PROGRAM Circuito_L8
VAR_INPUT
	Modo_Calibrar_L8: BOOL;
END_VAR
VAR
		fbBomba_L8 :Equipo_Motor_ATV320;
		ControlValv_ioLink_V1:ControlValv_ioLink;
		ControlValv_ioLink_V2: ControlValv_ioLink;
		ControlValv_ioLink_V3: ControlValv_ioLink;
		ControlValv_ioLink_V4: ControlValv_ioLink;
		Falla_L8_V1:BOOL;
		Falla_L8_V2:BOOL;
		Falla_L8_V3:BOOL;
		Falla_L8_V4:BOOL;
	Balanza_PU2_WT8: Balanza;
		dHS:DINT;
		TOF_calibradoIBC: TOF;
		PID_L8_SP:REAL;
		PID_L8_auto:BOOL;
		PID_L8_reset:BOOL;
		PID_L8_manual:REAL;
		PID_L8_bMuerta:REAL := 5;
		PID_L8_Kp:REAL := 0.1;
		PID_L8_Ti:REAL := 100;
		PID_L8_PV:REAL;
		Dosis_L8	:REAL;
		TiempoInyeccion_L8	:DINT;
		Peso	:REAL;
		Offset_L8:REAL;
		Inyeccion_L8:BOOL;
		Volumen_L8:REAL;
		Calculo_caudal_L8: Calculo_caudal;
		CorrecionCaudalxOffset_L8: CorrecionCaudalxOffset;
		tInyeccion: TON;
		Total :REAL;
		Totalant	:REAL;
		auxIniCal:BOOL;
		AuxVol:REAL;
		CA2_L8_V1_CmdA_Man :BOOL;
		CA2_L8_V4_CmdA_Man :BOOL;
		TDemoraInyectar: TON;
		SetDemoraInyeccion: REAL;
		Tiempo_seg_to_TIME_DemoraInyec: Tiempo_seg_to_TIME;
		AuxTDemoraInyec: TIME;
		PID_L8: FB_PID;		
		Tiempo_TIME_to_seg_InyCal: Tiempo_TIME_to_seg;
		AuxInyCal:TIME;	
		IniTotalFT2:REAL;
		Auxconsumo:REAL;
	ProductoAsociado: STRING;
	Lavagem_Circuito08: Lavagem;
	BasicPID_L8: FB_BasicPID;
	Teste: BOOL;
	Filtro:Filtro2;
	TON_StartBomba: TON;
END_VAR

VAR PERSISTENT
	UltimaCalibracao	:UDINT;	//Data e hora da ultima calibração
END_VAR
VAR // added by the converter: edge detectors and wires of the graphical bodies
    _w1, _w2, _w3, _w4, _w5, _w6, _w7, _w8, _w9, _w10, _w11, _w12, _w13 : BOOL;
    _ft1 : F_TRIG;
    _rt1, _rt2, _rt3 : R_TRIG;
END_VAR

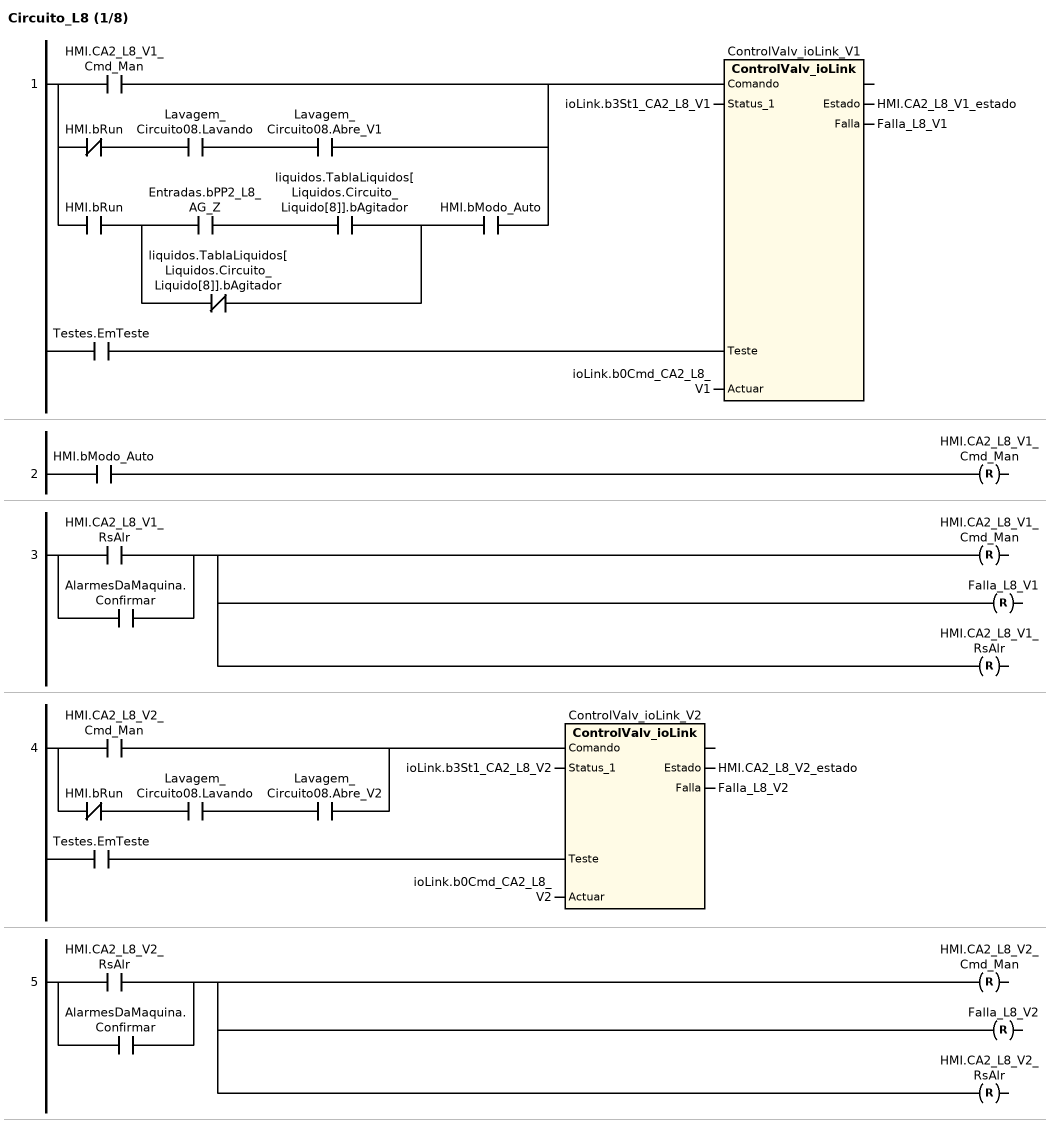
// NETWORK 1
ControlValv_ioLink_V1(
    Comando := HMI.CA2_L8_V1_Cmd_Man OR NOT HMI.bRun AND Lavagem_Circuito08.Lavando AND Lavagem_Circuito08.Abre_V1 OR HMI.bRun AND (Entradas.bPP2_L8_AG_Z AND (liquidos.TablaLiquidos[Liquidos.Circuito_Liquido[8]].bAgitador) OR NOT (liquidos.TablaLiquidos[Liquidos.Circuito_Liquido[8]].bAgitador)) AND HMI.bModo_Auto,
    Status_1 := ioLink.b3St1_CA2_L8_V1,
    Teste := Testes.EmTeste,
    Actuar := ioLink.b0Cmd_CA2_L8_V1,
    Estado => HMI.CA2_L8_V1_estado,
    Falla => Falla_L8_V1); // ControlValv_ioLink

// NETWORK 2
HMI.CA2_L8_V1_Cmd_Man R= HMI.bModo_Auto;

// NETWORK 3
_w1 := HMI.CA2_L8_V1_RsAlr OR AlarmesDaMaquina.Confirmar;
HMI.CA2_L8_V1_Cmd_Man R= _w1;
Falla_L8_V1 R= _w1;
HMI.CA2_L8_V1_RsAlr R= _w1;

// NETWORK 4
ControlValv_ioLink_V2(
    Comando := HMI.CA2_L8_V2_Cmd_Man OR NOT HMI.bRun AND Lavagem_Circuito08.Lavando AND Lavagem_Circuito08.Abre_V2,
    Status_1 := ioLink.b3St1_CA2_L8_V2,
    Teste := Testes.EmTeste,
    Actuar := ioLink.b0Cmd_CA2_L8_V2,
    Estado => HMI.CA2_L8_V2_estado,
    Falla => Falla_L8_V2); // ControlValv_ioLink

// NETWORK 5
_w2 := HMI.CA2_L8_V2_RsAlr OR AlarmesDaMaquina.Confirmar;
HMI.CA2_L8_V2_Cmd_Man R= _w2;
Falla_L8_V2 R= _w2;
HMI.CA2_L8_V2_RsAlr R= _w2;

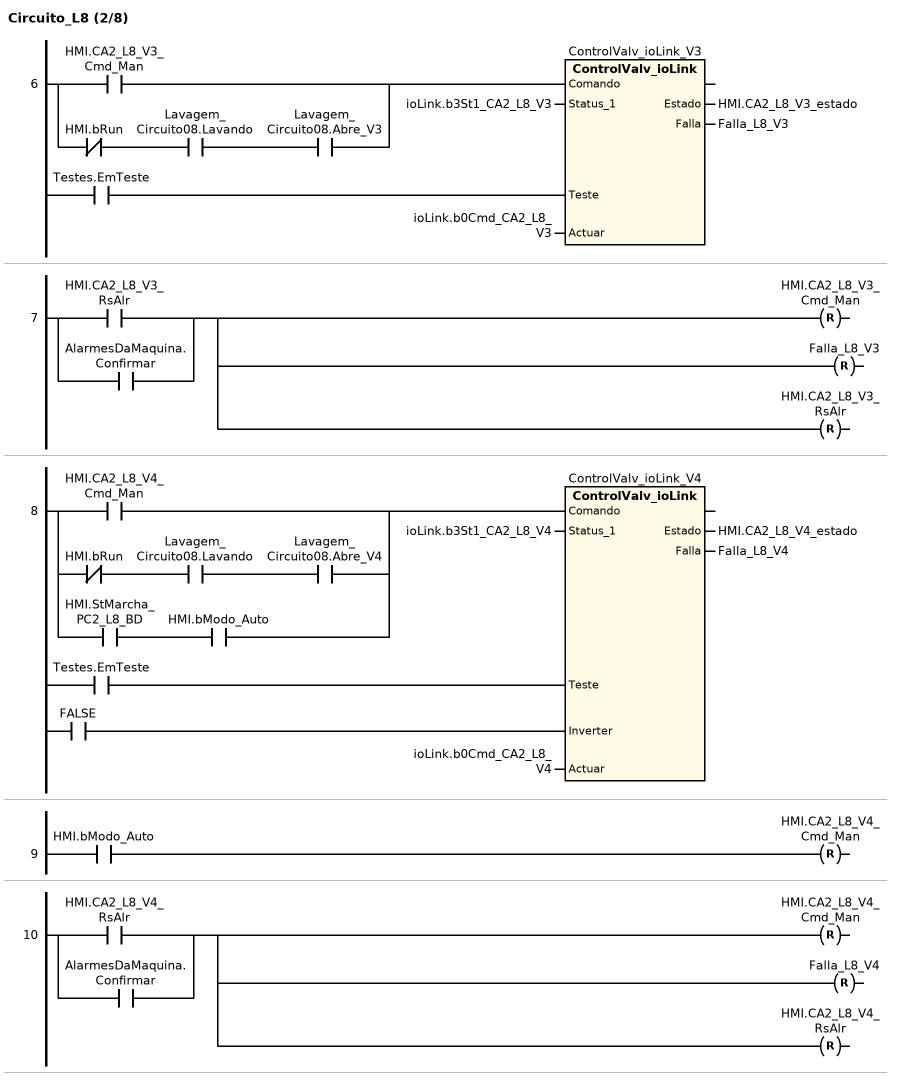
// NETWORK 6
ControlValv_ioLink_V3(
    Comando := HMI.CA2_L8_V3_Cmd_Man OR NOT HMI.bRun AND Lavagem_Circuito08.Lavando AND Lavagem_Circuito08.Abre_V3,
    Status_1 := ioLink.b3St1_CA2_L8_V3,
    Teste := Testes.EmTeste,
    Actuar := ioLink.b0Cmd_CA2_L8_V3,
    Estado => HMI.CA2_L8_V3_estado,
    Falla => Falla_L8_V3); // ControlValv_ioLink

// NETWORK 7
_w3 := HMI.CA2_L8_V3_RsAlr OR AlarmesDaMaquina.Confirmar;
HMI.CA2_L8_V3_Cmd_Man R= _w3;
Falla_L8_V3 R= _w3;
HMI.CA2_L8_V3_RsAlr R= _w3;

// NETWORK 8
ControlValv_ioLink_V4(
    Comando := HMI.CA2_L8_V4_Cmd_Man OR NOT HMI.bRun AND Lavagem_Circuito08.Lavando AND Lavagem_Circuito08.Abre_V4 OR HMI.StMarcha_PC2_L8_BD AND HMI.bModo_Auto,
    Status_1 := ioLink.b3St1_CA2_L8_V4,
    Teste := Testes.EmTeste,
    Inverter := FALSE,
    Actuar := ioLink.b0Cmd_CA2_L8_V4,
    Estado => HMI.CA2_L8_V4_estado,
    Falla => Falla_L8_V4); // ControlValv_ioLink

// NETWORK 9
HMI.CA2_L8_V4_Cmd_Man R= HMI.bModo_Auto;

// NETWORK 10
_w4 := HMI.CA2_L8_V4_RsAlr OR AlarmesDaMaquina.Confirmar;
HMI.CA2_L8_V4_Cmd_Man R= _w4;
Falla_L8_V4 R= _w4;
HMI.CA2_L8_V4_RsAlr R= _w4;

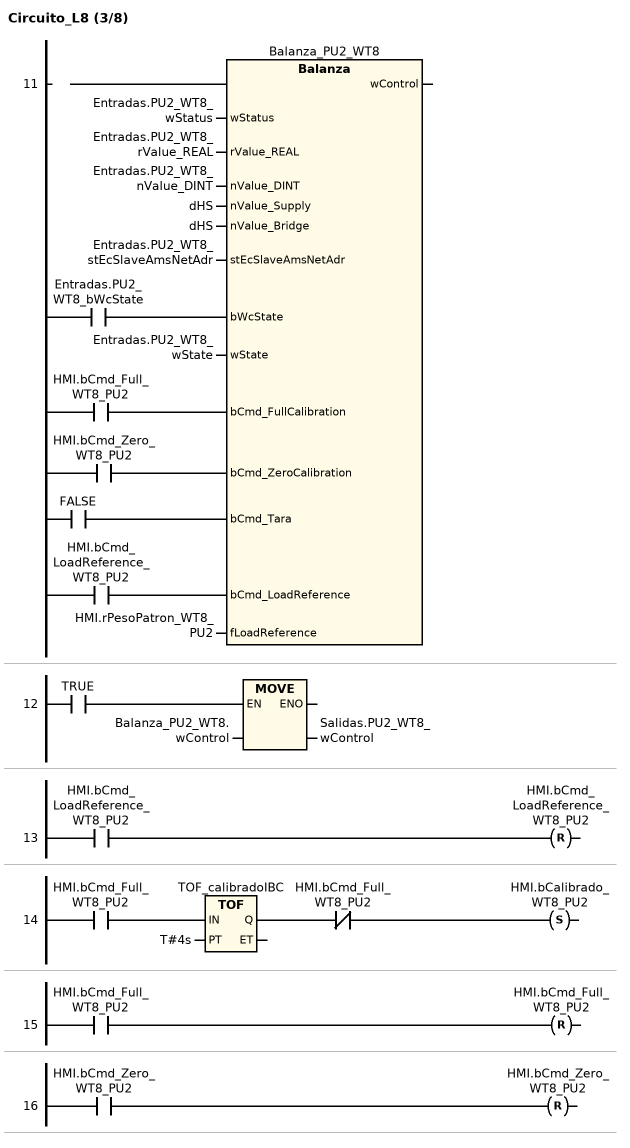
// NETWORK 11
Balanza_PU2_WT8(
    wStatus := Entradas.PU2_WT8_wStatus,
    rValue_REAL := Entradas.PU2_WT8_rValue_REAL,
    nValue_DINT := Entradas.PU2_WT8_nValue_DINT,
    nValue_Supply := dHS,
    nValue_Bridge := dHS,
    stEcSlaveAmsNetAdr := Entradas.PU2_WT8_stEcSlaveAmsNetAdr,
    bWcState := Entradas.PU2_WT8_bWcState,
    wState := Entradas.PU2_WT8_wState,
    bCmd_FullCalibration := HMI.bCmd_Full_WT8_PU2,
    bCmd_ZeroCalibration := HMI.bCmd_Zero_WT8_PU2,
    bCmd_Tara := FALSE,
    bCmd_LoadReference := HMI.bCmd_LoadReference_WT8_PU2,
    fLoadReference := HMI.rPesoPatron_WT8_PU2); // Balanza

// NETWORK 12
Salidas.PU2_WT8_wControl := Balanza_PU2_WT8.wControl;

// NETWORK 13
HMI.bCmd_LoadReference_WT8_PU2 R= HMI.bCmd_LoadReference_WT8_PU2;

// NETWORK 14
TOF_calibradoIBC(IN := HMI.bCmd_Full_WT8_PU2, PT := T#4s); // TOF
HMI.bCalibrado_WT8_PU2 S= TOF_calibradoIBC.Q AND NOT HMI.bCmd_Full_WT8_PU2;

// NETWORK 15
HMI.bCmd_Full_WT8_PU2 R= HMI.bCmd_Full_WT8_PU2;

// NETWORK 16
HMI.bCmd_Zero_WT8_PU2 R= HMI.bCmd_Zero_WT8_PU2;

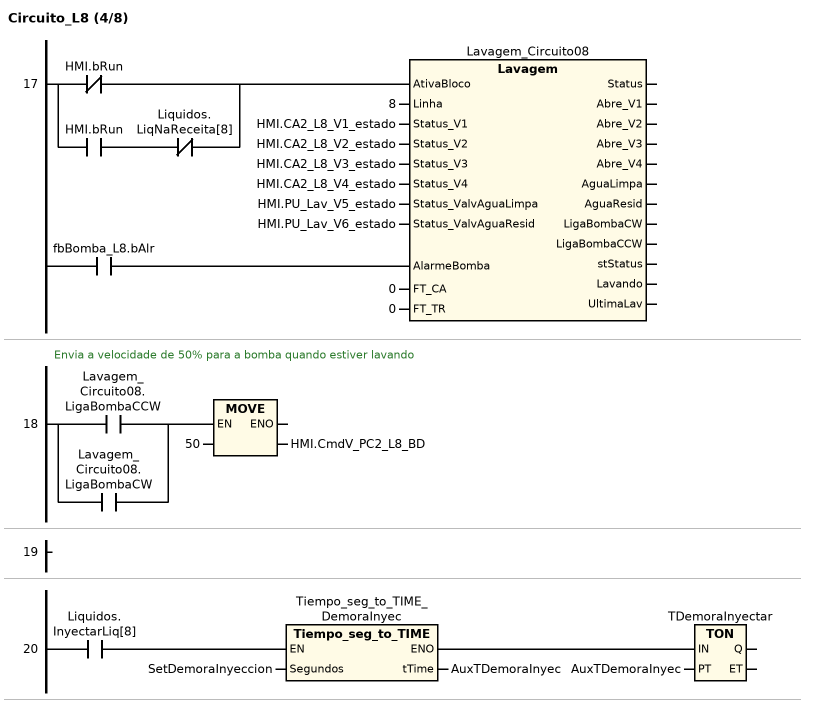
// NETWORK 17
Lavagem_Circuito08(
    AtivaBloco := NOT HMI.bRun OR HMI.bRun AND NOT Liquidos.LiqNaReceita[8],
    Linha := 8,
    Status_V1 := HMI.CA2_L8_V1_estado,
    Status_V2 := HMI.CA2_L8_V2_estado,
    Status_V3 := HMI.CA2_L8_V3_estado,
    Status_V4 := HMI.CA2_L8_V4_estado,
    Status_ValvAguaLimpa := HMI.PU_Lav_V5_estado,
    Status_ValvAguaResid := HMI.PU_Lav_V6_estado,
    AlarmeBomba := fbBomba_L8.bAlr,
    FT_CA := 0,
    FT_TR := 0); // Lavagem

// NETWORK 18
// Envia a velocidade de 50% para a bomba quando estiver lavando
IF Lavagem_Circuito08.LigaBombaCCW OR Lavagem_Circuito08.LigaBombaCW THEN HMI.CmdV_PC2_L8_BD := 50; END_IF

// NETWORK 19

// NETWORK 20
_w5 := Liquidos.InyectarLiq[8];
IF _w5 THEN
    Tiempo_seg_to_TIME_DemoraInyec(Segundos := SetDemoraInyeccion, tTime => AuxTDemoraInyec); // Tiempo_seg_to_TIME
END_IF
TDemoraInyectar(IN := _w5, PT := AuxTDemoraInyec); // TON

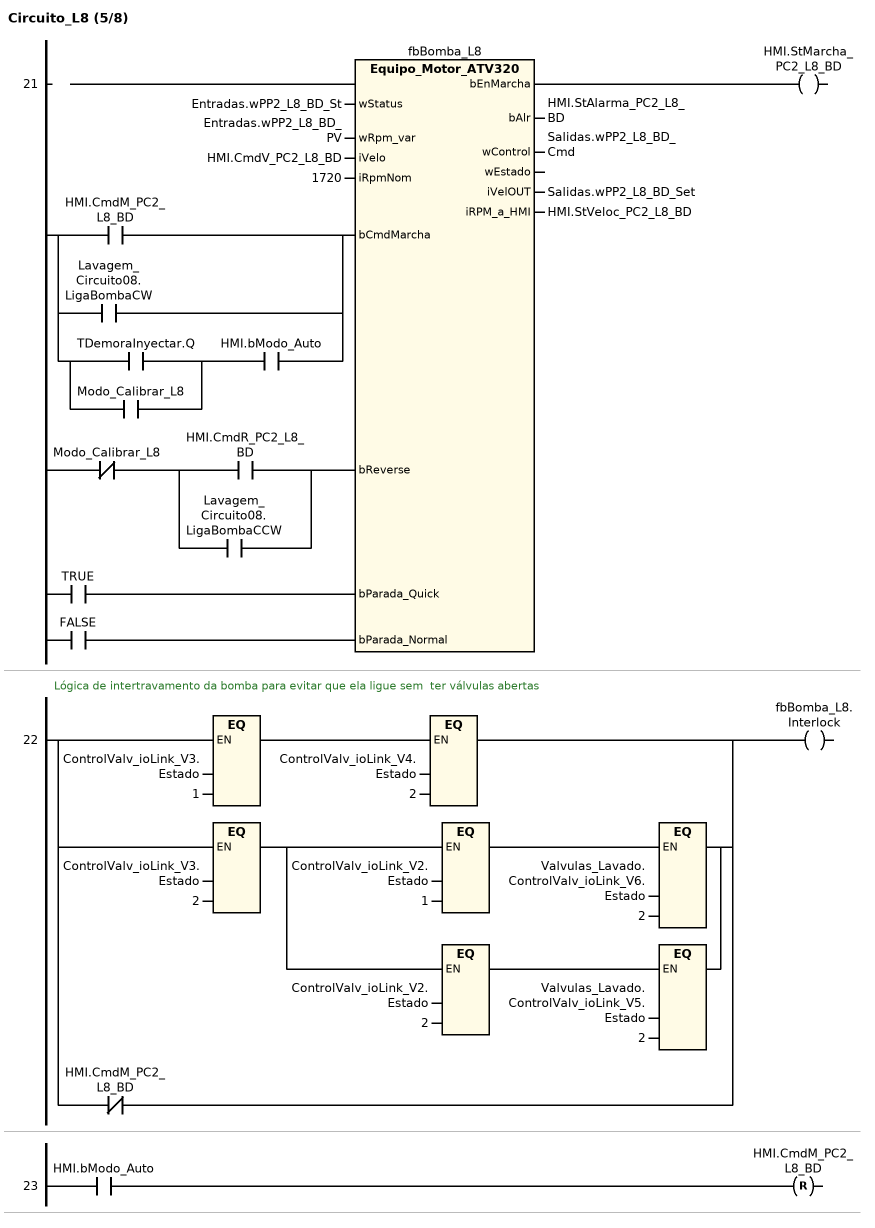
// NETWORK 21
fbBomba_L8(
    wStatus := Entradas.wPP2_L8_BD_St,
    wRpm_var := Entradas.wPP2_L8_BD_PV,
    iVelo := HMI.CmdV_PC2_L8_BD,
    iRpmNom := 1720,
    bCmdMarcha := HMI.CmdM_PC2_L8_BD OR Lavagem_Circuito08.LigaBombaCW OR (TDemoraInyectar.Q OR Modo_Calibrar_L8) AND HMI.bModo_Auto,
    bReverse := NOT Modo_Calibrar_L8 AND (HMI.CmdR_PC2_L8_BD OR Lavagem_Circuito08.LigaBombaCCW),
    bParada_Quick := TRUE,
    bParada_Normal := FALSE,
    bAlr => HMI.StAlarma_PC2_L8_BD,
    wControl => Salidas.wPP2_L8_BD_Cmd,
    iVelOUT => Salidas.wPP2_L8_BD_Set,
    iRPM_a_HMI => HMI.StVeloc_PC2_L8_BD); // Equipo_Motor_ATV320
HMI.StMarcha_PC2_L8_BD := fbBomba_L8.bEnMarcha;

// NETWORK 22
// Lógica de intertravamento da bomba para evitar que ela ligue sem  ter válvulas abertas
_w6 := NOT HMI.CmdM_PC2_L8_BD;
IF NOT _w6 THEN
    _w7 := ControlValv_ioLink_V3.Estado = 2;
    _w6 := ControlValv_ioLink_V3.Estado = 1 AND ControlValv_ioLink_V4.Estado = 2 OR (_w7 AND ControlValv_ioLink_V2.Estado = 1 AND Valvulas_Lavado.ControlValv_ioLink_V6.Estado = 2 OR _w7 AND ControlValv_ioLink_V2.Estado = 2 AND Valvulas_Lavado.ControlValv_ioLink_V5.Estado = 2);
END_IF
fbBomba_L8.Interlock := _w6;

// NETWORK 23
HMI.CmdM_PC2_L8_BD R= HMI.bModo_Auto;

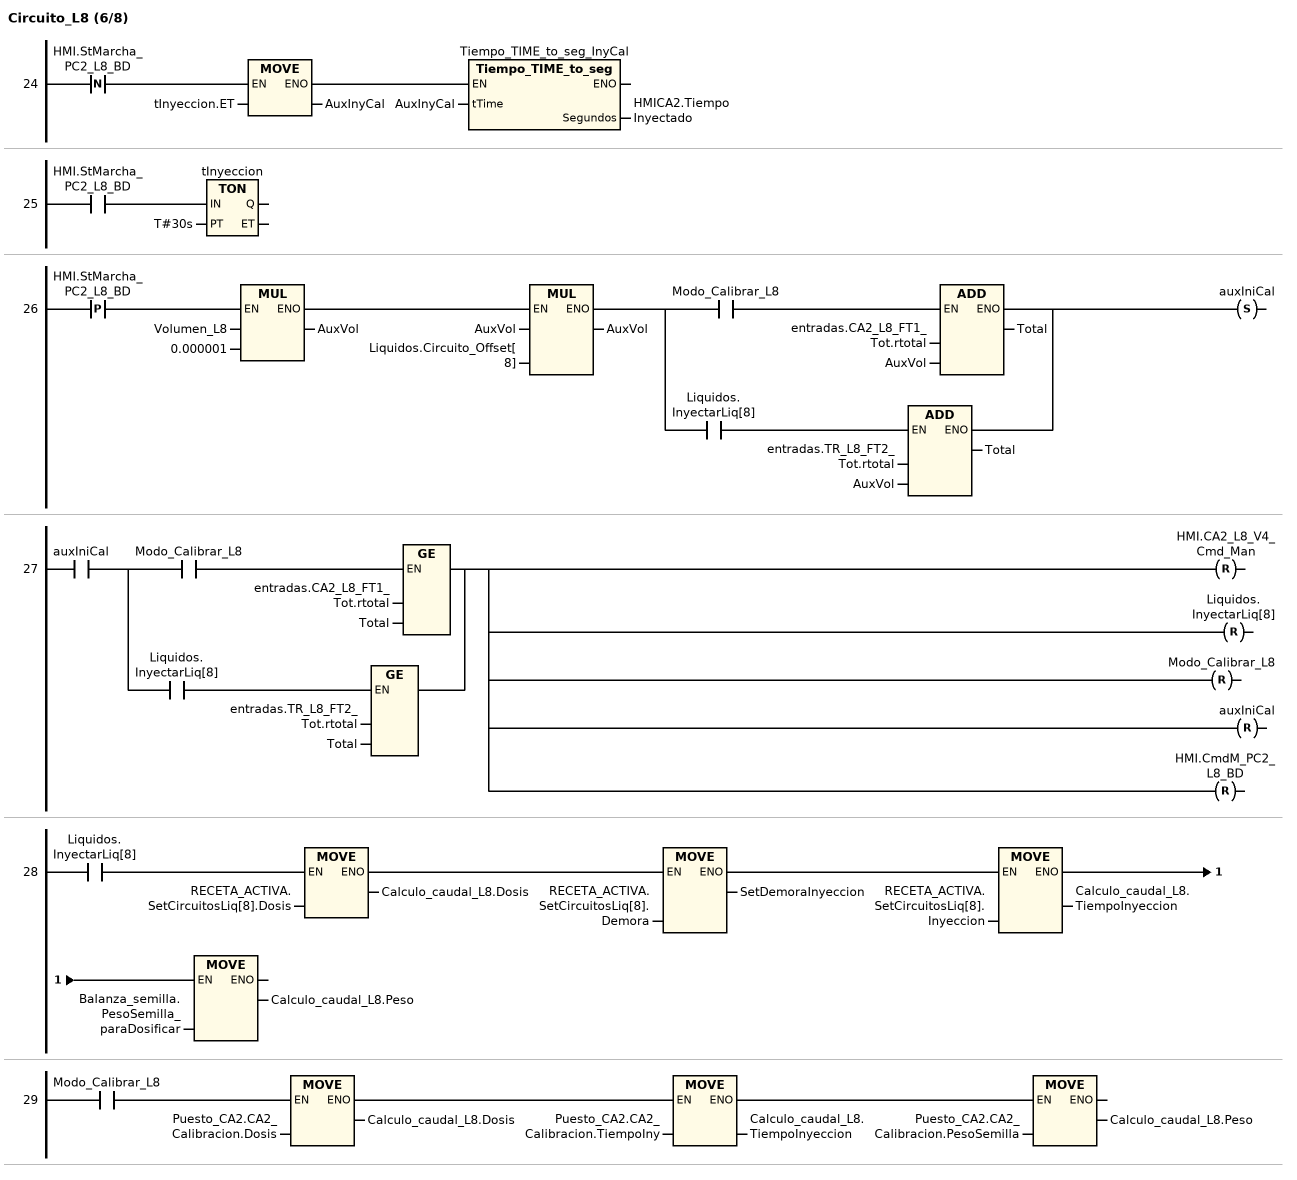
// NETWORK 24
_ft1(CLK := HMI.StMarcha_PC2_L8_BD);
_w8 := _ft1.Q;
IF _w8 THEN AuxInyCal := tInyeccion.ET; END_IF
IF _w8 THEN
    Tiempo_TIME_to_seg_InyCal(tTime := AuxInyCal, Segundos => HMICA2.TiempoInyectado); // Tiempo_TIME_to_seg
END_IF

// NETWORK 25
tInyeccion(IN := HMI.StMarcha_PC2_L8_BD, PT := T#30s); // TON

// NETWORK 26
_rt1(CLK := HMI.StMarcha_PC2_L8_BD);
_w9 := _rt1.Q;
IF _w9 THEN AuxVol := Volumen_L8 * 0.000001; END_IF
IF _w9 THEN AuxVol := AuxVol * Liquidos.Circuito_Offset[8]; END_IF
IF _w9 AND Modo_Calibrar_L8 THEN Total := entradas.CA2_L8_FT1_Tot.rtotal + AuxVol; END_IF
IF _w9 AND Liquidos.InyectarLiq[8] THEN Total := entradas.TR_L8_FT2_Tot.rtotal + AuxVol; END_IF
auxIniCal S= _w9 AND Modo_Calibrar_L8 OR _w9 AND Liquidos.InyectarLiq[8];

// NETWORK 27
_w10 := auxIniCal AND Modo_Calibrar_L8 AND entradas.CA2_L8_FT1_Tot.rtotal >= Total OR auxIniCal AND Liquidos.InyectarLiq[8] AND entradas.TR_L8_FT2_Tot.rtotal >= Total;
HMI.CA2_L8_V4_Cmd_Man R= _w10;
Liquidos.InyectarLiq[8] R= _w10;
Modo_Calibrar_L8 R= _w10;
auxIniCal R= _w10;
HMI.CmdM_PC2_L8_BD R= _w10;

// NETWORK 28
_w11 := Liquidos.InyectarLiq[8];
IF _w11 THEN Calculo_caudal_L8.Dosis := RECETA_ACTIVA.SetCircuitosLiq[8].Dosis; END_IF
IF _w11 THEN SetDemoraInyeccion := RECETA_ACTIVA.SetCircuitosLiq[8].Demora; END_IF
IF _w11 THEN Calculo_caudal_L8.TiempoInyeccion := RECETA_ACTIVA.SetCircuitosLiq[8].Inyeccion; END_IF
IF _w11 THEN Calculo_caudal_L8.Peso := Balanza_semilla.PesoSemilla_paraDosificar; END_IF

// NETWORK 29
_w12 := Modo_Calibrar_L8;
IF _w12 THEN Calculo_caudal_L8.Dosis := Puesto_CA2.CA2_Calibracion.Dosis; END_IF
IF _w12 THEN Calculo_caudal_L8.TiempoInyeccion := Puesto_CA2.CA2_Calibracion.TiempoIny; END_IF
IF _w12 THEN Calculo_caudal_L8.Peso := Puesto_CA2.CA2_Calibracion.PesoSemilla; END_IF

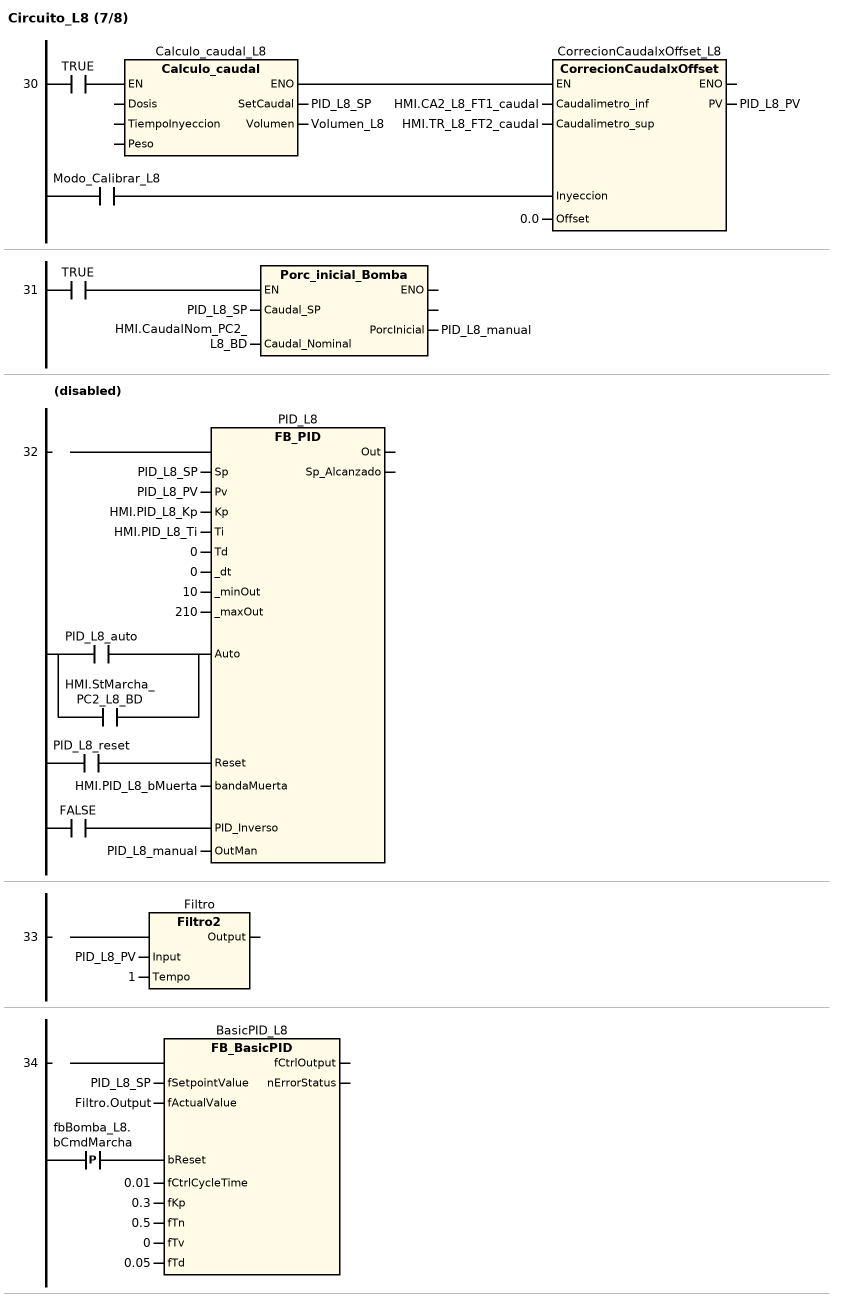
// NETWORK 30
Calculo_caudal_L8(SetCaudal => PID_L8_SP, Volumen => Volumen_L8); // Calculo_caudal
CorrecionCaudalxOffset_L8(
    Caudalimetro_inf := HMI.CA2_L8_FT1_caudal,
    Caudalimetro_sup := HMI.TR_L8_FT2_caudal,
    Inyeccion := Modo_Calibrar_L8,
    Offset := 0.0,
    PV => PID_L8_PV); // CorrecionCaudalxOffset

// NETWORK 31
Porc_inicial_Bomba(Caudal_SP := PID_L8_SP, Caudal_Nominal := HMI.CaudalNom_PC2_L8_BD, PorcInicial => PID_L8_manual);

// NETWORK 32 (disabled)
// PID_L8(
//     Sp := PID_L8_SP,
//     Pv := PID_L8_PV,
//     Kp := HMI.PID_L8_Kp,
//     Ti := HMI.PID_L8_Ti,
//     Td := 0,
//     _dt := 0,
//     _minOut := 10,
//     _maxOut := 210,
//     Auto := PID_L8_auto OR HMI.StMarcha_PC2_L8_BD,
//     Reset := PID_L8_reset,
//     bandaMuerta := HMI.PID_L8_bMuerta,
//     PID_Inverso := FALSE,
//     OutMan := PID_L8_manual); // FB_PID

// NETWORK 33
Filtro(Input := PID_L8_PV, Tempo := 1); // Filtro2

// NETWORK 34
_rt2(CLK := fbBomba_L8.bCmdMarcha);
BasicPID_L8(
    fSetpointValue := PID_L8_SP,
    fActualValue := Filtro.Output,
    bReset := _rt2.Q,
    fCtrlCycleTime := 0.01,
    fKp := 0.3,
    fTn := 0.5,
    fTv := 0,
    fTd := 0.05); // FB_BasicPID

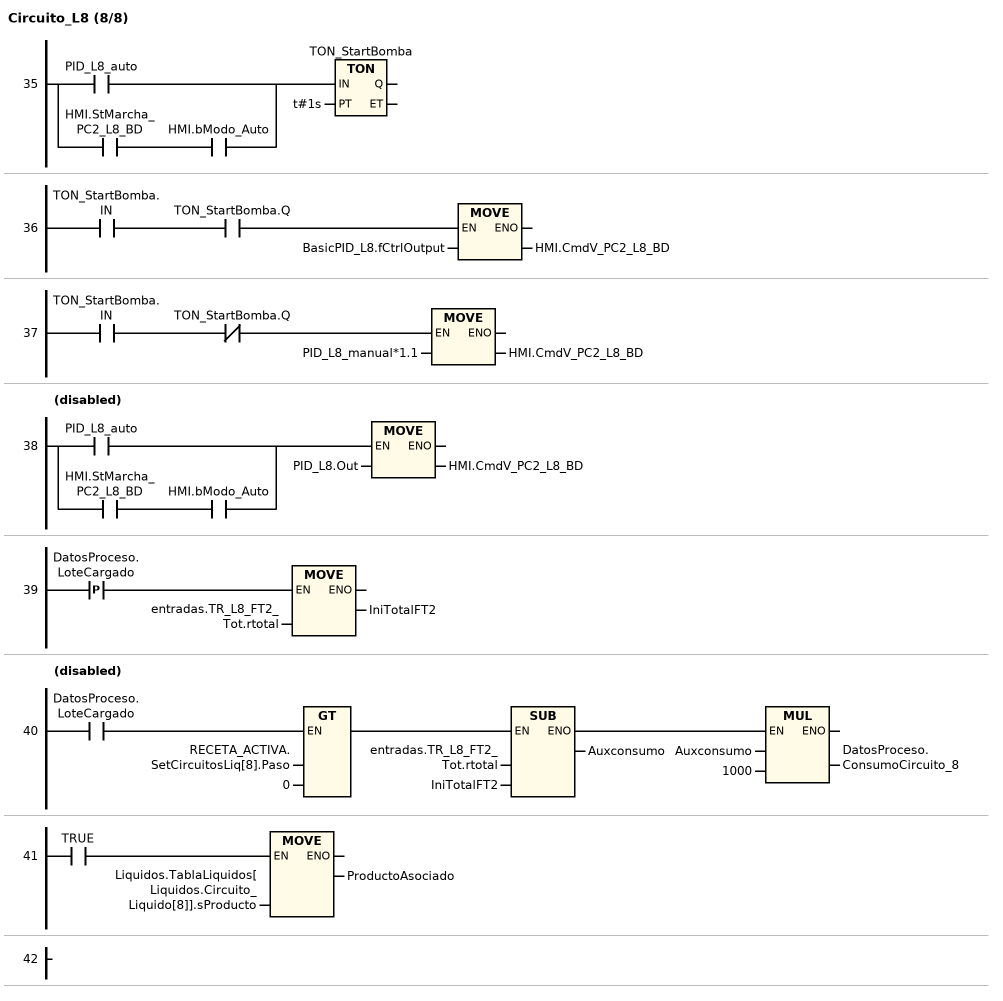
// NETWORK 35
TON_StartBomba(IN := PID_L8_auto OR HMI.StMarcha_PC2_L8_BD AND HMI.bModo_Auto, PT := t#1s); // TON

// NETWORK 36
IF TON_StartBomba.IN AND TON_StartBomba.Q THEN HMI.CmdV_PC2_L8_BD := BasicPID_L8.fCtrlOutput; END_IF

// NETWORK 37
IF TON_StartBomba.IN AND NOT TON_StartBomba.Q THEN HMI.CmdV_PC2_L8_BD := PID_L8_manual*1.1; END_IF

// NETWORK 38 (disabled)
// IF PID_L8_auto OR HMI.StMarcha_PC2_L8_BD AND HMI.bModo_Auto THEN HMI.CmdV_PC2_L8_BD := PID_L8.Out; END_IF

// NETWORK 39
_rt3(CLK := DatosProceso.LoteCargado);
IF _rt3.Q THEN IniTotalFT2 := entradas.TR_L8_FT2_Tot.rtotal; END_IF

// NETWORK 40 (disabled)
// _w13 := DatosProceso.LoteCargado AND RECETA_ACTIVA.SetCircuitosLiq[8].Paso > 0;
// IF _w13 THEN Auxconsumo := entradas.TR_L8_FT2_Tot.rtotal - IniTotalFT2; END_IF
// IF _w13 THEN DatosProceso.ConsumoCircuito_8 := Auxconsumo * 1000; END_IF

// NETWORK 41
ProductoAsociado := Liquidos.TablaLiquidos[Liquidos.Circuito_Liquido[8]].sProducto;

// NETWORK 42

END_PROGRAM

(* stored: Version 1.1.0.1, ProductVersion 3.1.4024.14
   POU Circuito_L8: Id {56db3373-50e6-4018-b318-2ad379db81a1}, SpecialFunc None *)
